FUNCTION_BLOCK ConveyorCTLServer (* Basic Function Block Type *)
  (* Standard: 61499-2 *)
  (* Version 0.2, 2003-12-04, JHC, Rockwell Automation, Renamed for better indexing. *)
  (* Version 0.1, 2002-11-05, JHC, Rockwell Automation, Corrected missing ST element in Algorithm REQ. *)
  (* Version 0.0, 2000-05-30, JHC, Rockwell Automation *)
  (* Compiler header: package fb.rt.cs725; *)
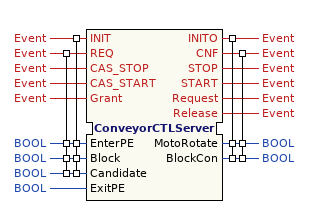
  EVENT_INPUT
    INIT WITH EnterPE, Block, Candidate; (* Initialization Request *)
    REQ WITH EnterPE, Block, Candidate; (* Normal Execution Request *)
    CAS_STOP;
    CAS_START;
    Grant;
  END_EVENT
  EVENT_OUTPUT
    INITO WITH MotoRotate, BlockCon; (* Initialization Confirm *)
    CNF WITH MotoRotate, BlockCon; (* Execution Confirmation *)
    STOP;
    START;
    Request;
    Release;
  END_EVENT
  VAR_INPUT
    EnterPE : BOOL; (* Input event qualifier *)
    Block : BOOL;
    Candidate : BOOL;
    ExitPE : BOOL;
  END_VAR
  VAR_OUTPUT
    MotoRotate : BOOL; (* Output event qualifier *)
    BlockCon : BOOL;
  END_VAR
  VAR
    lastPE : BOOL := 1;
    lastBlock : BOOL := 0;
  END_VAR
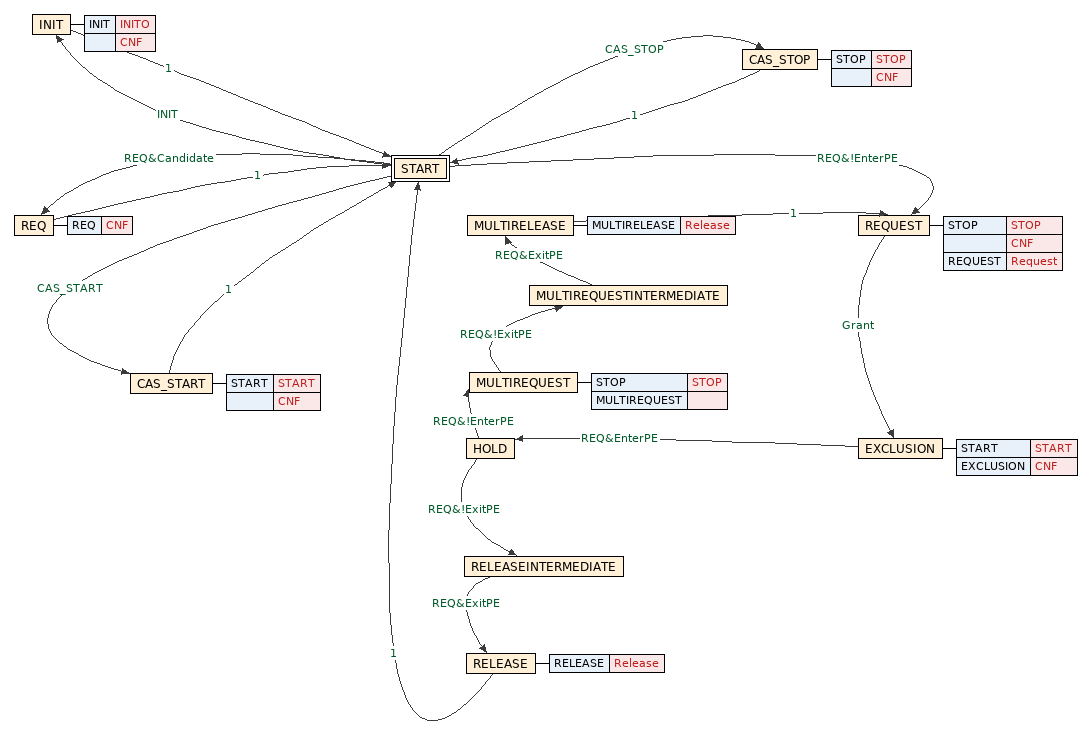
  EC_STATES
    START; (* Initial State *)
    INIT : INIT -> INITO, -> CNF; (* Initialization *)
    REQ : REQ -> CNF; (* Normal execution *)
    CAS_START : START -> START, -> CNF;
    CAS_STOP : STOP -> STOP, -> CNF;
    REQUEST : STOP -> STOP, -> CNF, REQUEST -> Request;
    EXCLUSION : START -> START, EXCLUSION -> CNF;
    RELEASE : RELEASE -> Release;
    HOLD;
    MULTIREQUEST : STOP -> STOP, MULTIREQUEST;
    MULTIRELEASE : MULTIRELEASE -> Release;
    RELEASEINTERMEDIATE;
    MULTIREQUESTINTERMEDIATE;
  END_STATES
  EC_TRANSITIONS
    START TO INIT := INIT;
    INIT TO START := 1;
    START TO REQ := REQ&Candidate;
    REQ TO START := 1;
    START TO CAS_START := CAS_START;
    CAS_START TO START := 1;
    START TO CAS_STOP := CAS_STOP;
    CAS_STOP TO START := 1;
    REQUEST TO EXCLUSION := Grant;
    HOLD TO RELEASEINTERMEDIATE := REQ&!ExitPE;
    RELEASE TO START := 1;
    START TO REQUEST := REQ&!EnterPE;
    EXCLUSION TO HOLD := REQ&EnterPE;
    HOLD TO MULTIREQUEST := REQ&!EnterPE;
    MULTIREQUEST TO MULTIREQUESTINTERMEDIATE := REQ&!ExitPE;
    MULTIRELEASE TO REQUEST := 1;
    RELEASEINTERMEDIATE TO RELEASE := REQ&ExitPE;
    MULTIREQUESTINTERMEDIATE TO MULTIRELEASE := REQ&ExitPE;
  END_TRANSITIONS
  ALGORITHM INIT IN ST: (* Initialization algorithm *)
MotoRotate := TRUE;
Block := FALSE;

System.out.println(this + " " + MotoRotate);
System.out.println(MotoRotate);
  END_ALGORITHM
  ALGORITHM REQ IN ST: (* Normally executed algorithm *)
System.out.println(this +  " -> Candidate" + Candidate);
IF Candidate THEN
IF lastPE !:= EnterPE THEN
IF NOT EnterPE THEN
BlockCon:= TRUE;
System.out.println("BlockCon = true");
ELSE
BlockCon:=FALSE;
System.out.println("BlockCon = false");
END_IF
lastPE := EnterPE;
END_IF
IF lastBlock !:= Block THEN
IF Block THEN
STOP.serviceEvent(this);
MotoRotate := FALSE;
System.out.println("Cas Stop");
ELSE
START.serviceEvent(this);
MotoRotate := TRUE;
System.out.println("Cas Start");
END_IF
lastBlock := Block;
END_IF
END_IF
  END_ALGORITHM
  ALGORITHM START IN ST:
MotoRotate:=TRUE;
System.out.println(this + " Start " + MotoRotate);

System.out.println("Start " + MotoRotate);
  END_ALGORITHM
  ALGORITHM STOP IN Java:
MotoRotate.value=false;
System.out.println(this+" Stop "+MotoRotate.value);

System.out.println("Stop "+MotoRotate.value);
  END_ALGORITHM
  ALGORITHM REQUEST IN Java:
System.out.println("Entered Request state: " + this);
  END_ALGORITHM
  ALGORITHM EXCLUSION IN Java:
System.out.println("Entered Exclusion state");
  END_ALGORITHM
  ALGORITHM MULTIREQUEST IN Java:
System.out.println("Entered Multirequest state");
  END_ALGORITHM
  ALGORITHM MULTIRELEASE IN Java:
System.out.println("Entered multirelease state");
  END_ALGORITHM
  ALGORITHM RELEASE IN Java:
System.out.println("Entered Release state");
  END_ALGORITHM
END_FUNCTION_BLOCK
